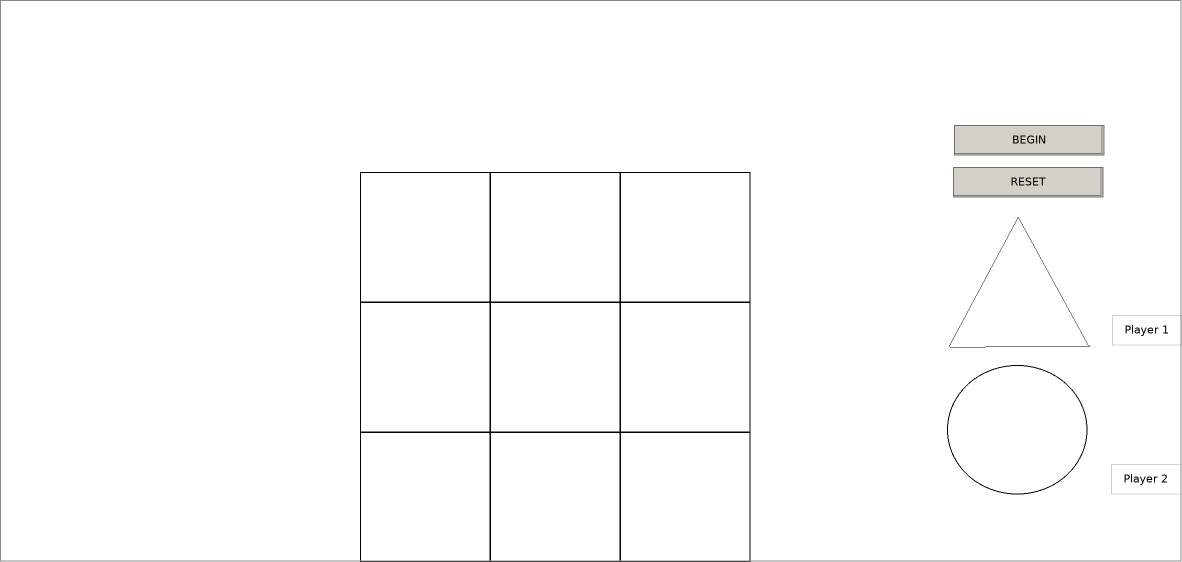
VISUALIZATION Visualization  // 1182x562
    Rectangle (360,172 130x130)
        tap GVL.Rechthoek_1
    Rectangle (490,172 130x130)
        tap GVL.Rechthoek_2
    Rectangle (620,172 130x130)
        tap GVL.Rechthoek_3
    Rectangle (360,302 130x130)
        tap GVL.Rechthoek_4
    Rectangle (490,302 130x130)
        tap GVL.Rechthoek_5
    Rectangle (620,302 130x130)
        tap GVL.Rechthoek_6
    Rectangle (360,432 130x130)
        tap GVL.Rechthoek_7
    Rectangle (490,432 130x130)
        tap GVL.Rechthoek_8
    Rectangle (620,432 130x130)
        tap GVL.Rechthoek_9
    Textfield (1112,315 70x30), "Player 1"
    Textfield (1111,464 70x30), "Player 2"
    Button (954,125 150x30), "BEGIN"
        tap GVL.Begin_Knop
    Polygon (949,346) (1018,217) (1088,345) (1090,346) (950,347), colour toggle: GVL.Player_1_Lamp
    Ellipse (947,365 140x129), colour toggle: GVL.Player_2_Lamp
    Button (953,167 150x30), "RESET"
        tap GVL.Reset_Knop
    Ellipse (363,175 125x125), colour toggle: GVL.Rondje_1
        tap GVL.Rechthoek_1
    Ellipse (493,175 125x125), colour toggle: GVL.Rondje_2
        tap GVL.Rechthoek_2
    Ellipse (623,175 125x125), colour toggle: GVL.Rondje_3
        tap GVL.Rechthoek_3
    Ellipse (623,305 125x125), colour toggle: GVL.Rondje_6
        tap GVL.Rechthoek_6
    Ellipse (493,305 125x125), colour toggle: GVL.Rondje_5
        tap GVL.Rechthoek_5
    Ellipse (363,305 125x125), colour toggle: GVL.Rondje_4
        tap GVL.Rechthoek_4
    Ellipse (363,435 125x125), colour toggle: GVL.Rondje_7
        tap GVL.Rechthoek_7
    Ellipse (493,435 125x125), colour toggle: GVL.Rondje_8
        tap GVL.Rechthoek_8
    Ellipse (623,435 125x125), colour toggle: GVL.Rondje_9
        tap GVL.Rechthoek_9
    Polygon (363,297) (428,177) (488,297) (488,297) (363,297), colour toggle: GVL.Driehoek_1
        tap GVL.Rechthoek_1
    Polygon (493,297) (558,177) (618,297) (618,297) (493,297), colour toggle: GVL.Driehoek_2
        tap GVL.Rechthoek_2
    Polygon (623,297) (688,177) (748,297) (748,297) (623,297), colour toggle: GVL.Driehoek_3
        tap GVL.Rechthoek_3
    Polygon (623,427) (688,307) (748,427) (748,427) (623,427), colour toggle: GVL.Driehoek_6
        tap GVL.Rechthoek_6
    Polygon (493,427) (558,307) (618,427) (618,427) (493,427), colour toggle: GVL.Driehoek_5
        tap GVL.Rechthoek_5
    Polygon (363,427) (428,307) (488,427) (488,427) (363,427), colour toggle: GVL.Driehoek_4
        tap GVL.Rechthoek_4
    Polygon (623,557) (688,437) (748,557) (748,557) (623,557), colour toggle: GVL.Driehoek_9
        tap GVL.Rechthoek_9
    Polygon (493,557) (558,437) (618,557) (618,557) (493,557), colour toggle: GVL.Driehoek_8
        tap GVL.Rechthoek_8
    Polygon (363,557) (428,437) (488,557) (488,557) (363,557), colour toggle: GVL.Driehoek_7
        tap GVL.Rechthoek_7
END_VISUALIZATION

(* stored: Version 1.1.0.1, ProductVersion 3.1.4024.12
   Visu Visualization: Id {3ba9bd90-6832-4c1d-a352-2fb7a9ec481e} *)
